// TIA Portal V20 export
// export: Created 2025-12-01T14:57:00.8344037Z, ExportSetting None, DisplayName Totally Integrated Automation Portal, DisplayVersion V20 Update 3, DisplayName TIA Portal Openness, DisplayVersion V20 Update 3, DisplayName TIA Portal Version Control Interface, DisplayVersion V20 Update 3, DisplayName STEP 7 Professional, DisplayVersion V20 Update 3, DisplayName STEP 7 Safety, DisplayVersion V20 Update 2, DisplayName WinCC Basic/Comfort/Advanced, DisplayVersion V20 Update 3, DisplayName WinCC Professional, DisplayVersion V20 Update 3, DisplayName WinCC Unified, DisplayVersion V20 Update 3
FUNCTION "FC455_TL_TR_E1_S2_Aus" : Void   // FC455, LAD
{ S7_Optimized_Access := 'FALSE' }
AUTHOR : TLigero
NAME : 20160208
VERSION : 3.5
// stored: AutoNumber false, SetENOAutomatically false
   VAR_INPUT
      Mesa : UInt;
      En_Tension : Bool;
      pHsMx_E1 : Bool;
      pHsMx_S2 : Bool;
      Termico_E1_Tx : Bool;
      Termico_S2_Tx : Bool;
      Avance_E1_Tx_Ok : Bool;
      Avance_S2_Tx_Ok : Bool;
      PosTR_E1 : Bool;
      PosTR_S2 : Bool;
      AVTF_MAnt_Mx : Bool;
      PTF_Mx_MSig : Bool;
      NXT_Avance : Bool;
      V_CNT_ApHsMx_E1 : UDInt;
      V_CNT_ApHsMx_S2 : UDInt;
      V_Paro : UDInt;
      V_TOut_Tx_Mx : UDInt;
      V_TOut_TR : UDInt;
   END_VAR
   VAR_OUTPUT
      PTF_MAnt_Mx : Bool;
      AVTF_Mx_MSig : Bool;
      NXT_Descarga_Act : Bool;
   END_VAR
   VAR_IN_OUT
      MAux_FN_Phs_E1 : Bool;
      Maux_FN_Phs_S2 : Bool;
      Mem_FN_phs_E1 : Bool;
      Mem_FN_phs_S2 : Bool;
   END_VAR
   VAR_TEMP
      Mem_CNT_Aus_Ent : Bool;
      OK_VACIADO : Bool;
      Mem_CNT_Aus_Sal : Bool;
      Aux_Parar : Bool;
      tout_atasco : Bool;
      tout_transfer : Bool;
      Mem_CNT_Tmp_Paro_Tx : Bool;
      TEMP_MA_TR_Pos_E1 : Bool;
      TEMP_MA_TR_Pos_S2 : Bool;
      ok_tension : Bool;
   END_VAR
   VAR_TEMP   // added for the SCL form of the ladder/FBD networks
      _w1 : Bool;
      _w2 : Bool;
   END_VAR
BEGIN

REGION Network 1: Marca General Error
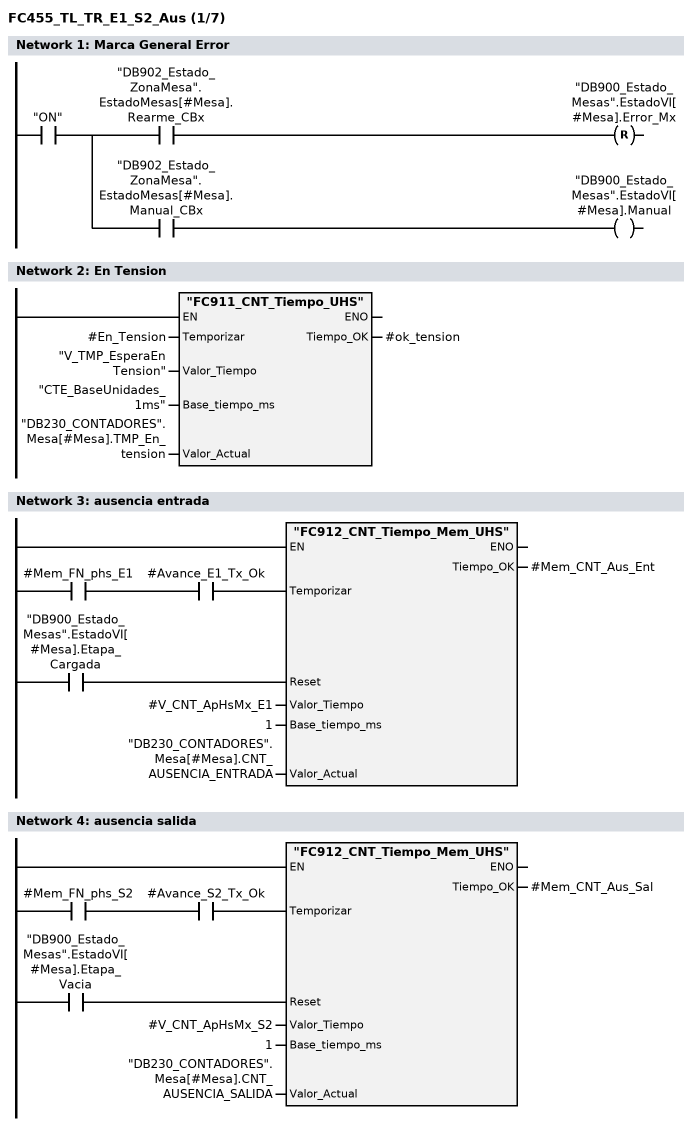
   RUNG wire#powerrail
      Contact( "ON" )
      wire#w1
      Contact( "DB902_Estado_ZonaMesa".EstadoMesas[#Mesa].Rearme_CBx )
      R_Coil( "DB900_Estado_Mesas".EstadoVI[#Mesa].Error_Mx )
   END_RUNG
   RUNG wire#w1
      Contact( "DB902_Estado_ZonaMesa".EstadoMesas[#Mesa].Manual_CBx )
      Coil( "DB900_Estado_Mesas".EstadoVI[#Mesa].Manual )
   END_RUNG
   // the same network as SCL:
   IF "ON" AND "DB902_Estado_ZonaMesa".EstadoMesas[#Mesa].Rearme_CBx THEN
       "DB900_Estado_Mesas".EstadoVI[#Mesa].Error_Mx := FALSE;
   END_IF;
   "DB900_Estado_Mesas".EstadoVI[#Mesa].Manual := "ON" AND "DB902_Estado_ZonaMesa".EstadoMesas[#Mesa].Manual_CBx;
END_REGION

REGION Network 2: En Tension
   RUNG wire#powerrail
      "FC911_CNT_Tiempo_UHS"(Temporizar := #En_Tension, Valor_Tiempo := "V_TMP_EsperaEnTension", Base_tiempo_ms := "CTE_BaseUnidades_1ms", Valor_Actual := "DB230_CONTADORES".Mesa[#Mesa].TMP_En_tension, Tiempo_OK => #ok_tension)
   END_RUNG
   // the same network as SCL:
   "FC911_CNT_Tiempo_UHS"(Temporizar := #En_Tension,
                          Valor_Tiempo := "V_TMP_EsperaEnTension",
                          Base_tiempo_ms := "CTE_BaseUnidades_1ms",
                          Valor_Actual := "DB230_CONTADORES".Mesa[#Mesa].TMP_En_tension,
                          Tiempo_OK => #ok_tension);
END_REGION

REGION Network 3: ausencia entrada
   RUNG wire#powerrail
      "FC912_CNT_Tiempo_Mem_UHS"(Temporizar := wire#w1, Reset := wire#w2, Valor_Tiempo := #V_CNT_ApHsMx_E1, Base_tiempo_ms := 1, Valor_Actual := "DB230_CONTADORES".Mesa[#Mesa].CNT_AUSENCIA_ENTRADA, Tiempo_OK => #Mem_CNT_Aus_Ent)
   END_RUNG
   RUNG wire#powerrail
      Contact( #Mem_FN_phs_E1 )
      Contact( #Avance_E1_Tx_Ok )
   END_RUNG wire#w1
   RUNG wire#powerrail
      Contact( "DB900_Estado_Mesas".EstadoVI[#Mesa].Etapa_Cargada )
   END_RUNG wire#w2
   // the same network as SCL:
   "FC912_CNT_Tiempo_Mem_UHS"(Temporizar := #Mem_FN_phs_E1 AND #Avance_E1_Tx_Ok,
                           Reset := "DB900_Estado_Mesas".EstadoVI[#Mesa].Etapa_Cargada,
                           Valor_Tiempo := #V_CNT_ApHsMx_E1,
                           Base_tiempo_ms := 1,
                           Valor_Actual := "DB230_CONTADORES".Mesa[#Mesa].CNT_AUSENCIA_ENTRADA,
                           Tiempo_OK => #Mem_CNT_Aus_Ent);
END_REGION

REGION Network 4: ausencia salida
   RUNG wire#powerrail
      "FC912_CNT_Tiempo_Mem_UHS"(Temporizar := wire#w1, Reset := wire#w2, Valor_Tiempo := #V_CNT_ApHsMx_S2, Base_tiempo_ms := 1, Valor_Actual := "DB230_CONTADORES".Mesa[#Mesa].CNT_AUSENCIA_SALIDA, Tiempo_OK => #Mem_CNT_Aus_Sal)
   END_RUNG
   RUNG wire#powerrail
      Contact( #Mem_FN_phs_S2 )
      Contact( #Avance_S2_Tx_Ok )
   END_RUNG wire#w1
   RUNG wire#powerrail
      Contact( "DB900_Estado_Mesas".EstadoVI[#Mesa].Etapa_Vacia )
   END_RUNG wire#w2
   // the same network as SCL:
   "FC912_CNT_Tiempo_Mem_UHS"(Temporizar := #Mem_FN_phs_S2 AND #Avance_S2_Tx_Ok,
                           Reset := "DB900_Estado_Mesas".EstadoVI[#Mesa].Etapa_Vacia,
                           Valor_Tiempo := #V_CNT_ApHsMx_S2,
                           Base_tiempo_ms := 1,
                           Valor_Actual := "DB230_CONTADORES".Mesa[#Mesa].CNT_AUSENCIA_SALIDA,
                           Tiempo_OK => #Mem_CNT_Aus_Sal);
END_REGION

REGION Network 5: MEMORIAS DE FLANCOS
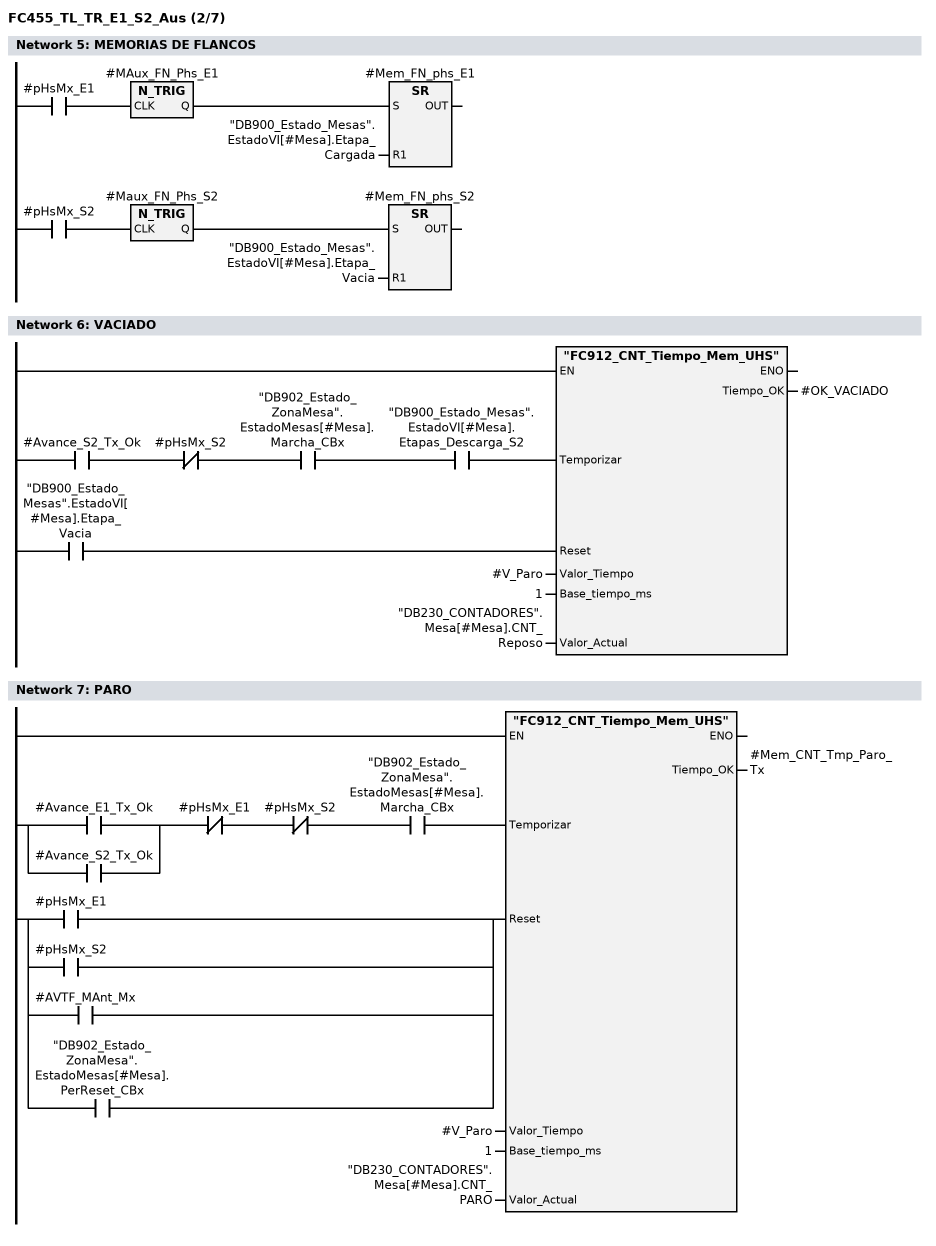
   RUNG wire#powerrail
      Contact( #pHsMx_E1 )
      N_Trig( #MAux_FN_Phs_E1 )
      S_SR(operand := #Mem_FN_phs_E1, r1 := "DB900_Estado_Mesas".EstadoVI[#Mesa].Etapa_Cargada)
   END_RUNG
   RUNG wire#powerrail
      Contact( #pHsMx_S2 )
      N_Trig( #Maux_FN_Phs_S2 )
      S_SR(operand := #Mem_FN_phs_S2, r1 := "DB900_Estado_Mesas".EstadoVI[#Mesa].Etapa_Vacia)
   END_RUNG
   // the same network as SCL:
   #_w1 := NOT #pHsMx_E1 AND #MAux_FN_Phs_E1;   // falling edge
   #MAux_FN_Phs_E1 := #pHsMx_E1;
   IF #_w1 THEN
       #Mem_FN_phs_E1 := TRUE;   // SR flip-flop
   END_IF;
   IF "DB900_Estado_Mesas".EstadoVI[#Mesa].Etapa_Cargada THEN #Mem_FN_phs_E1 := FALSE; END_IF;
   #_w2 := NOT #pHsMx_S2 AND #Maux_FN_Phs_S2;   // falling edge
   #Maux_FN_Phs_S2 := #pHsMx_S2;
   IF #_w2 THEN
       #Mem_FN_phs_S2 := TRUE;   // SR flip-flop
   END_IF;
   IF "DB900_Estado_Mesas".EstadoVI[#Mesa].Etapa_Vacia THEN #Mem_FN_phs_S2 := FALSE; END_IF;
END_REGION

REGION Network 6: VACIADO
   RUNG wire#powerrail
      "FC912_CNT_Tiempo_Mem_UHS"(Temporizar := wire#w1, Reset := wire#w2, Valor_Tiempo := #V_Paro, Base_tiempo_ms := 1, Valor_Actual := "DB230_CONTADORES".Mesa[#Mesa].CNT_Reposo, Tiempo_OK => #OK_VACIADO)
   END_RUNG
   RUNG wire#powerrail
      Contact( #Avance_S2_Tx_Ok )
      I_Contact( #pHsMx_S2 )
      Contact( "DB902_Estado_ZonaMesa".EstadoMesas[#Mesa].Marcha_CBx )
      Contact( "DB900_Estado_Mesas".EstadoVI[#Mesa].Etapas_Descarga_S2 )
   END_RUNG wire#w1
   RUNG wire#powerrail
      Contact( "DB900_Estado_Mesas".EstadoVI[#Mesa].Etapa_Vacia )
   END_RUNG wire#w2
   // the same network as SCL:
   "FC912_CNT_Tiempo_Mem_UHS"(Temporizar := #Avance_S2_Tx_Ok AND NOT #pHsMx_S2 AND "DB902_Estado_ZonaMesa".EstadoMesas[#Mesa].Marcha_CBx AND "DB900_Estado_Mesas".EstadoVI[#Mesa].Etapas_Descarga_S2,
                           Reset := "DB900_Estado_Mesas".EstadoVI[#Mesa].Etapa_Vacia,
                           Valor_Tiempo := #V_Paro,
                           Base_tiempo_ms := 1,
                           Valor_Actual := "DB230_CONTADORES".Mesa[#Mesa].CNT_Reposo,
                           Tiempo_OK => #OK_VACIADO);
END_REGION

REGION Network 7: PARO
   RUNG wire#powerrail
      "FC912_CNT_Tiempo_Mem_UHS"(Temporizar := wire#w2, Reset := wire#w3, Valor_Tiempo := #V_Paro, Base_tiempo_ms := 1, Valor_Actual := "DB230_CONTADORES".Mesa[#Mesa].CNT_PARO, Tiempo_OK => #Mem_CNT_Tmp_Paro_Tx)
   END_RUNG
   RUNG wire#powerrail
      Contact( #Avance_E1_Tx_Ok )
      wire#w1
      I_Contact( #pHsMx_E1 )
      I_Contact( #pHsMx_S2 )
      Contact( "DB902_Estado_ZonaMesa".EstadoMesas[#Mesa].Marcha_CBx )
   END_RUNG wire#w2
   RUNG wire#powerrail
      Contact( #Avance_S2_Tx_Ok )
   END_RUNG wire#w1
   RUNG wire#powerrail
      Contact( #pHsMx_E1 )
   END_RUNG wire#w3
   RUNG wire#powerrail
      Contact( #pHsMx_S2 )
   END_RUNG wire#w3
   RUNG wire#powerrail
      Contact( #AVTF_MAnt_Mx )
   END_RUNG wire#w3
   RUNG wire#powerrail
      Contact( "DB902_Estado_ZonaMesa".EstadoMesas[#Mesa].PerReset_CBx )
   END_RUNG wire#w3
   // the same network as SCL:
   "FC912_CNT_Tiempo_Mem_UHS"(Temporizar := (#Avance_E1_Tx_Ok OR #Avance_S2_Tx_Ok) AND NOT #pHsMx_E1 AND NOT #pHsMx_S2 AND "DB902_Estado_ZonaMesa".EstadoMesas[#Mesa].Marcha_CBx,
                           Reset := #pHsMx_E1 OR #pHsMx_S2 OR #AVTF_MAnt_Mx OR "DB902_Estado_ZonaMesa".EstadoMesas[#Mesa].PerReset_CBx,
                           Valor_Tiempo := #V_Paro,
                           Base_tiempo_ms := 1,
                           Valor_Actual := "DB230_CONTADORES".Mesa[#Mesa].CNT_PARO,
                           Tiempo_OK => #Mem_CNT_Tmp_Paro_Tx);
END_REGION

REGION Network 8: Etapa MESA CARGADA
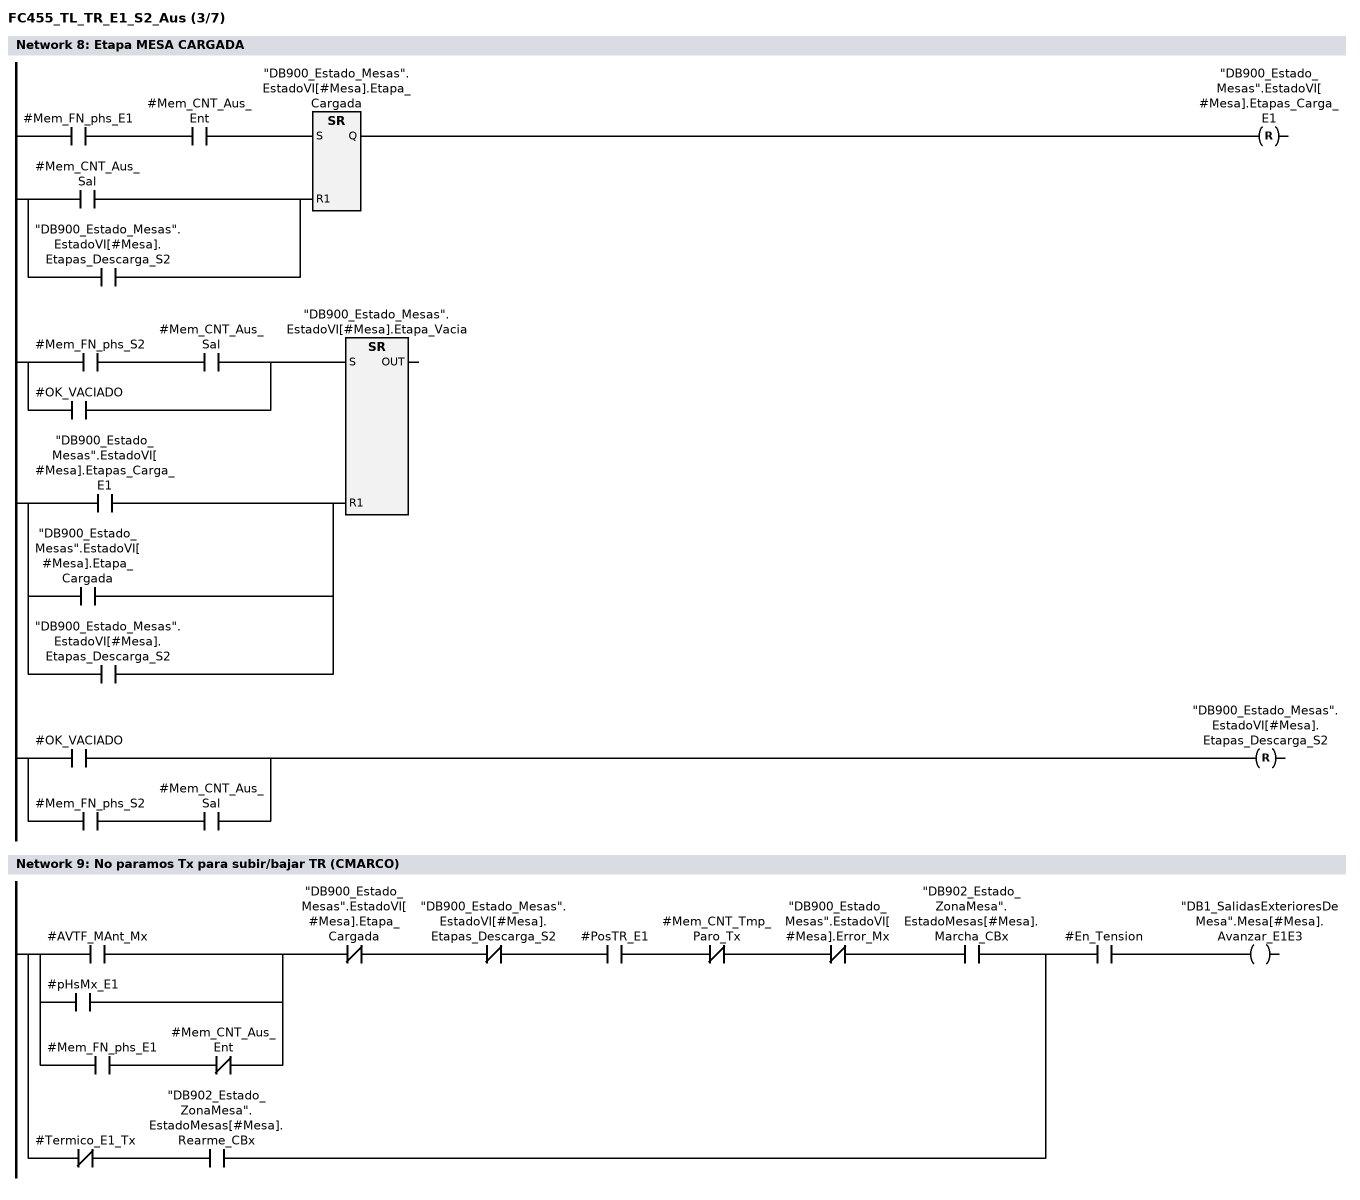
   RUNG wire#powerrail
      Contact( #Mem_FN_phs_E1 )
      Contact( #Mem_CNT_Aus_Ent )
      S_SR(operand := "DB900_Estado_Mesas".EstadoVI[#Mesa].Etapa_Cargada, r1 := wire#w1)
      R_Coil( "DB900_Estado_Mesas".EstadoVI[#Mesa].Etapas_Carga_E1 )
   END_RUNG
   RUNG wire#powerrail
      Contact( #Mem_CNT_Aus_Sal )
   END_RUNG wire#w1
   RUNG wire#powerrail
      Contact( "DB900_Estado_Mesas".EstadoVI[#Mesa].Etapas_Descarga_S2 )
   END_RUNG wire#w1
   RUNG wire#powerrail
      Contact( #Mem_FN_phs_S2 )
      Contact( #Mem_CNT_Aus_Sal )
      wire#w2
      S_SR(operand := "DB900_Estado_Mesas".EstadoVI[#Mesa].Etapa_Vacia, r1 := wire#w3)
   END_RUNG
   RUNG wire#powerrail
      Contact( #OK_VACIADO )
   END_RUNG wire#w2
   RUNG wire#powerrail
      Contact( "DB900_Estado_Mesas".EstadoVI[#Mesa].Etapas_Carga_E1 )
   END_RUNG wire#w3
   RUNG wire#powerrail
      Contact( "DB900_Estado_Mesas".EstadoVI[#Mesa].Etapa_Cargada )
   END_RUNG wire#w3
   RUNG wire#powerrail
      Contact( "DB900_Estado_Mesas".EstadoVI[#Mesa].Etapas_Descarga_S2 )
   END_RUNG wire#w3
   RUNG wire#powerrail
      Contact( #OK_VACIADO )
      wire#w4
      R_Coil( "DB900_Estado_Mesas".EstadoVI[#Mesa].Etapas_Descarga_S2 )
   END_RUNG
   RUNG wire#powerrail
      Contact( #Mem_FN_phs_S2 )
      Contact( #Mem_CNT_Aus_Sal )
   END_RUNG wire#w4
   // the same network as SCL:
   #_w1 := #Mem_CNT_Aus_Sal OR "DB900_Estado_Mesas".EstadoVI[#Mesa].Etapas_Descarga_S2;
   IF #Mem_FN_phs_E1 AND #Mem_CNT_Aus_Ent THEN
       "DB900_Estado_Mesas".EstadoVI[#Mesa].Etapa_Cargada := TRUE;   // SR flip-flop
   END_IF;
   IF #_w1 THEN "DB900_Estado_Mesas".EstadoVI[#Mesa].Etapa_Cargada := FALSE; END_IF;
   IF "DB900_Estado_Mesas".EstadoVI[#Mesa].Etapa_Cargada THEN
       "DB900_Estado_Mesas".EstadoVI[#Mesa].Etapas_Carga_E1 := FALSE;
   END_IF;
   #_w2 := "DB900_Estado_Mesas".EstadoVI[#Mesa].Etapas_Carga_E1 OR "DB900_Estado_Mesas".EstadoVI[#Mesa].Etapa_Cargada OR "DB900_Estado_Mesas".EstadoVI[#Mesa].Etapas_Descarga_S2;
   IF (#Mem_FN_phs_S2 AND #Mem_CNT_Aus_Sal) OR #OK_VACIADO THEN
       "DB900_Estado_Mesas".EstadoVI[#Mesa].Etapa_Vacia := TRUE;   // SR flip-flop
   END_IF;
   IF #_w2 THEN "DB900_Estado_Mesas".EstadoVI[#Mesa].Etapa_Vacia := FALSE; END_IF;
   IF #OK_VACIADO OR (#Mem_FN_phs_S2 AND #Mem_CNT_Aus_Sal) THEN
       "DB900_Estado_Mesas".EstadoVI[#Mesa].Etapas_Descarga_S2 := FALSE;
   END_IF;
END_REGION

REGION Network 9: No paramos Tx para subir/bajar TR (CMARCO)
   RUNG wire#powerrail
      Contact( #AVTF_MAnt_Mx )
      wire#w1
      I_Contact( "DB900_Estado_Mesas".EstadoVI[#Mesa].Etapa_Cargada )
      I_Contact( "DB900_Estado_Mesas".EstadoVI[#Mesa].Etapas_Descarga_S2 )
      Contact( #PosTR_E1 )
      I_Contact( #Mem_CNT_Tmp_Paro_Tx )
      I_Contact( "DB900_Estado_Mesas".EstadoVI[#Mesa].Error_Mx )
      Contact( "DB902_Estado_ZonaMesa".EstadoMesas[#Mesa].Marcha_CBx )
      wire#w2
      Contact( #En_Tension )
      Coil( "DB1_SalidasExterioresDeMesa".Mesa[#Mesa].Avanzar_E1E3 )
   END_RUNG
   RUNG wire#powerrail
      Contact( #pHsMx_E1 )
   END_RUNG wire#w1
   RUNG wire#powerrail
      Contact( #Mem_FN_phs_E1 )
      I_Contact( #Mem_CNT_Aus_Ent )
   END_RUNG wire#w1
   RUNG wire#powerrail
      I_Contact( #Termico_E1_Tx )
      Contact( "DB902_Estado_ZonaMesa".EstadoMesas[#Mesa].Rearme_CBx )
   END_RUNG wire#w2
   // the same network as SCL:
   "DB1_SalidasExterioresDeMesa".Mesa[#Mesa].Avanzar_E1E3 := (((#AVTF_MAnt_Mx OR #pHsMx_E1 OR (#Mem_FN_phs_E1 AND NOT #Mem_CNT_Aus_Ent)) AND NOT "DB900_Estado_Mesas".EstadoVI[#Mesa].Etapa_Cargada AND NOT "DB900_Estado_Mesas".EstadoVI[#Mesa].Etapas_Descarga_S2 AND #PosTR_E1 AND NOT #Mem_CNT_Tmp_Paro_Tx AND NOT "DB900_Estado_Mesas".EstadoVI[#Mesa].Error_Mx AND "DB902_Estado_ZonaMesa".EstadoMesas[#Mesa].Marcha_CBx) OR (NOT #Termico_E1_Tx AND "DB902_Estado_ZonaMesa".EstadoMesas[#Mesa].Rearme_CBx)) AND #En_Tension;
END_REGION

REGION Network 10: Quito el forzar paroTx (MA 02/06/08)
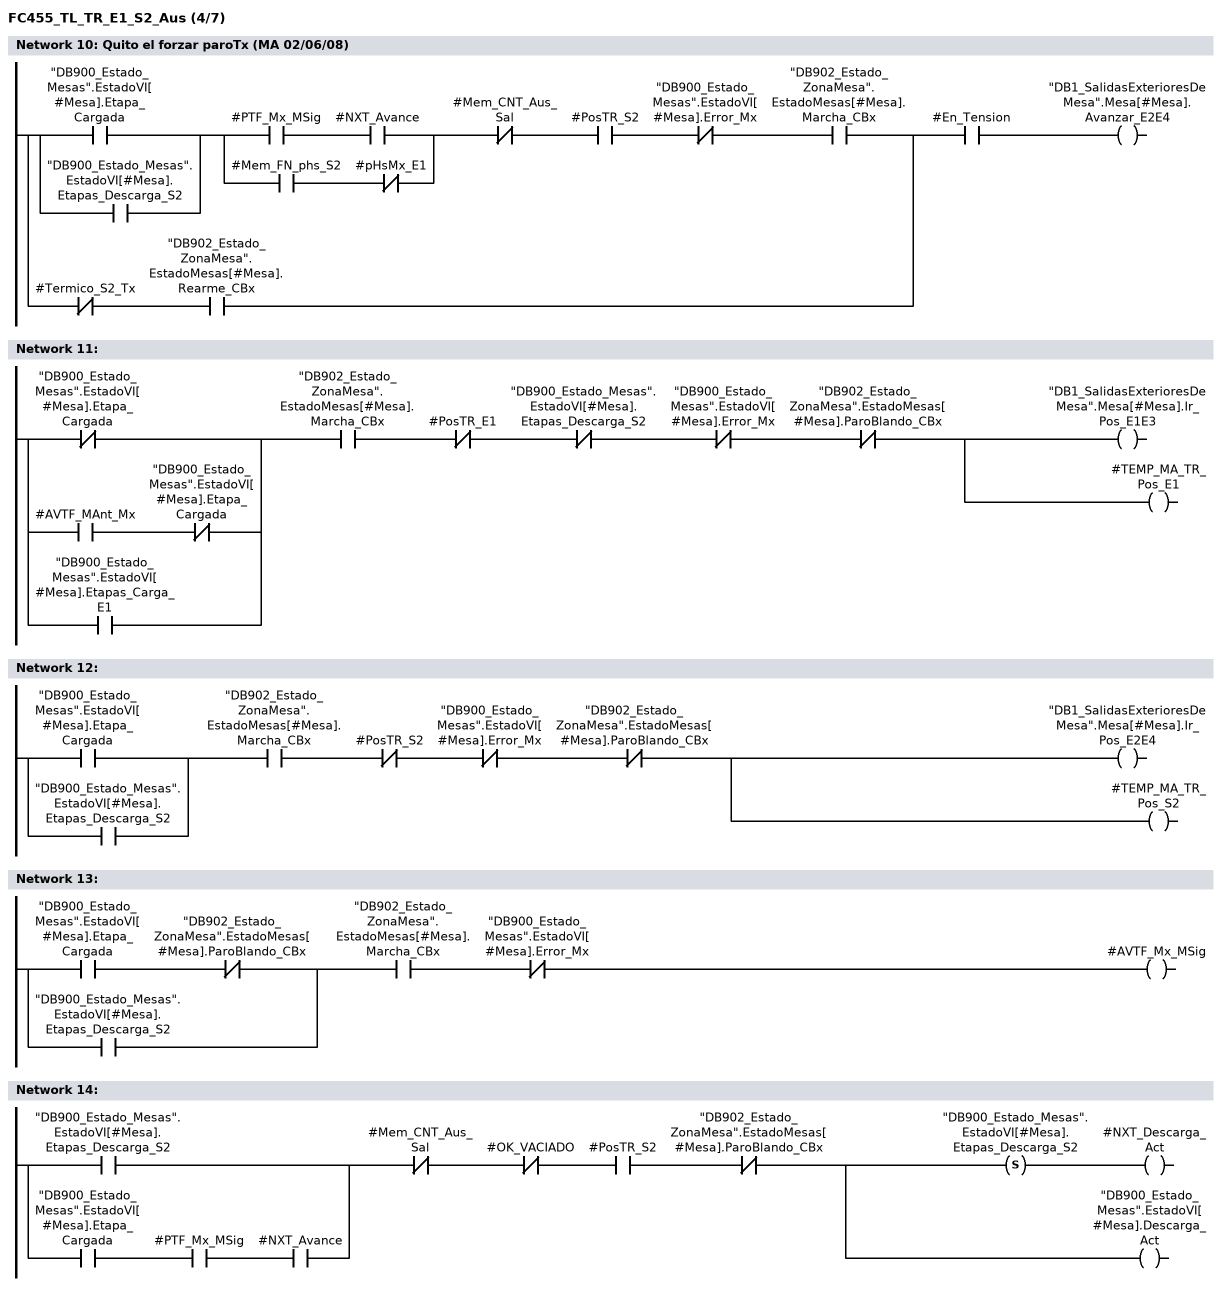
   RUNG wire#powerrail
      Contact( "DB900_Estado_Mesas".EstadoVI[#Mesa].Etapa_Cargada )
      wire#w1
      Contact( #PTF_Mx_MSig )
      Contact( #NXT_Avance )
      wire#w2
      I_Contact( #Mem_CNT_Aus_Sal )
      Contact( #PosTR_S2 )
      I_Contact( "DB900_Estado_Mesas".EstadoVI[#Mesa].Error_Mx )
      Contact( "DB902_Estado_ZonaMesa".EstadoMesas[#Mesa].Marcha_CBx )
      wire#w3
      Contact( #En_Tension )
      Coil( "DB1_SalidasExterioresDeMesa".Mesa[#Mesa].Avanzar_E2E4 )
   END_RUNG
   RUNG wire#powerrail
      Contact( "DB900_Estado_Mesas".EstadoVI[#Mesa].Etapas_Descarga_S2 )
   END_RUNG wire#w1
   RUNG wire#w1
      Contact( #Mem_FN_phs_S2 )
      I_Contact( #pHsMx_E1 )
   END_RUNG wire#w2
   RUNG wire#powerrail
      I_Contact( #Termico_S2_Tx )
      Contact( "DB902_Estado_ZonaMesa".EstadoMesas[#Mesa].Rearme_CBx )
   END_RUNG wire#w3
   // the same network as SCL:
   "DB1_SalidasExterioresDeMesa".Mesa[#Mesa].Avanzar_E2E4 := ((("DB900_Estado_Mesas".EstadoVI[#Mesa].Etapa_Cargada OR "DB900_Estado_Mesas".EstadoVI[#Mesa].Etapas_Descarga_S2) AND ((#PTF_Mx_MSig AND #NXT_Avance) OR (#Mem_FN_phs_S2 AND NOT #pHsMx_E1)) AND NOT #Mem_CNT_Aus_Sal AND #PosTR_S2 AND NOT "DB900_Estado_Mesas".EstadoVI[#Mesa].Error_Mx AND "DB902_Estado_ZonaMesa".EstadoMesas[#Mesa].Marcha_CBx) OR (NOT #Termico_S2_Tx AND "DB902_Estado_ZonaMesa".EstadoMesas[#Mesa].Rearme_CBx)) AND #En_Tension;
END_REGION

REGION Network 11
   RUNG wire#powerrail
      I_Contact( "DB900_Estado_Mesas".EstadoVI[#Mesa].Etapa_Cargada )
      wire#w1
      Contact( "DB902_Estado_ZonaMesa".EstadoMesas[#Mesa].Marcha_CBx )
      I_Contact( #PosTR_E1 )
      I_Contact( "DB900_Estado_Mesas".EstadoVI[#Mesa].Etapas_Descarga_S2 )
      I_Contact( "DB900_Estado_Mesas".EstadoVI[#Mesa].Error_Mx )
      I_Contact( "DB902_Estado_ZonaMesa".EstadoMesas[#Mesa].ParoBlando_CBx )
      wire#w2
      Coil( "DB1_SalidasExterioresDeMesa".Mesa[#Mesa].Ir_Pos_E1E3 )
   END_RUNG
   RUNG wire#powerrail
      Contact( #AVTF_MAnt_Mx )
      I_Contact( "DB900_Estado_Mesas".EstadoVI[#Mesa].Etapa_Cargada )
   END_RUNG wire#w1
   RUNG wire#powerrail
      Contact( "DB900_Estado_Mesas".EstadoVI[#Mesa].Etapas_Carga_E1 )
   END_RUNG wire#w1
   RUNG wire#w2
      Coil( #TEMP_MA_TR_Pos_E1 )
   END_RUNG
   // the same network as SCL:
   #_w1 := (NOT "DB900_Estado_Mesas".EstadoVI[#Mesa].Etapa_Cargada OR (#AVTF_MAnt_Mx AND NOT "DB900_Estado_Mesas".EstadoVI[#Mesa].Etapa_Cargada) OR "DB900_Estado_Mesas".EstadoVI[#Mesa].Etapas_Carga_E1) AND "DB902_Estado_ZonaMesa".EstadoMesas[#Mesa].Marcha_CBx AND NOT #PosTR_E1 AND NOT "DB900_Estado_Mesas".EstadoVI[#Mesa].Etapas_Descarga_S2 AND NOT "DB900_Estado_Mesas".EstadoVI[#Mesa].Error_Mx AND NOT "DB902_Estado_ZonaMesa".EstadoMesas[#Mesa].ParoBlando_CBx;
   "DB1_SalidasExterioresDeMesa".Mesa[#Mesa].Ir_Pos_E1E3 := (NOT "DB900_Estado_Mesas".EstadoVI[#Mesa].Etapa_Cargada OR (#AVTF_MAnt_Mx AND NOT "DB900_Estado_Mesas".EstadoVI[#Mesa].Etapa_Cargada) OR "DB900_Estado_Mesas".EstadoVI[#Mesa].Etapas_Carga_E1) AND "DB902_Estado_ZonaMesa".EstadoMesas[#Mesa].Marcha_CBx AND NOT #PosTR_E1 AND NOT "DB900_Estado_Mesas".EstadoVI[#Mesa].Etapas_Descarga_S2 AND NOT "DB900_Estado_Mesas".EstadoVI[#Mesa].Error_Mx AND NOT "DB902_Estado_ZonaMesa".EstadoMesas[#Mesa].ParoBlando_CBx;
   #TEMP_MA_TR_Pos_E1 := #_w1;
END_REGION

REGION Network 12
   RUNG wire#powerrail
      Contact( "DB900_Estado_Mesas".EstadoVI[#Mesa].Etapa_Cargada )
      wire#w1
      Contact( "DB902_Estado_ZonaMesa".EstadoMesas[#Mesa].Marcha_CBx )
      I_Contact( #PosTR_S2 )
      I_Contact( "DB900_Estado_Mesas".EstadoVI[#Mesa].Error_Mx )
      I_Contact( "DB902_Estado_ZonaMesa".EstadoMesas[#Mesa].ParoBlando_CBx )
      wire#w2
      Coil( "DB1_SalidasExterioresDeMesa".Mesa[#Mesa].Ir_Pos_E2E4 )
   END_RUNG
   RUNG wire#powerrail
      Contact( "DB900_Estado_Mesas".EstadoVI[#Mesa].Etapas_Descarga_S2 )
   END_RUNG wire#w1
   RUNG wire#w2
      Coil( #TEMP_MA_TR_Pos_S2 )
   END_RUNG
   // the same network as SCL:
   #_w1 := ("DB900_Estado_Mesas".EstadoVI[#Mesa].Etapa_Cargada OR "DB900_Estado_Mesas".EstadoVI[#Mesa].Etapas_Descarga_S2) AND "DB902_Estado_ZonaMesa".EstadoMesas[#Mesa].Marcha_CBx AND NOT #PosTR_S2 AND NOT "DB900_Estado_Mesas".EstadoVI[#Mesa].Error_Mx AND NOT "DB902_Estado_ZonaMesa".EstadoMesas[#Mesa].ParoBlando_CBx;
   "DB1_SalidasExterioresDeMesa".Mesa[#Mesa].Ir_Pos_E2E4 := ("DB900_Estado_Mesas".EstadoVI[#Mesa].Etapa_Cargada OR "DB900_Estado_Mesas".EstadoVI[#Mesa].Etapas_Descarga_S2) AND "DB902_Estado_ZonaMesa".EstadoMesas[#Mesa].Marcha_CBx AND NOT #PosTR_S2 AND NOT "DB900_Estado_Mesas".EstadoVI[#Mesa].Error_Mx AND NOT "DB902_Estado_ZonaMesa".EstadoMesas[#Mesa].ParoBlando_CBx;
   #TEMP_MA_TR_Pos_S2 := #_w1;
END_REGION

REGION Network 13
   RUNG wire#powerrail
      Contact( "DB900_Estado_Mesas".EstadoVI[#Mesa].Etapa_Cargada )
      I_Contact( "DB902_Estado_ZonaMesa".EstadoMesas[#Mesa].ParoBlando_CBx )
      wire#w1
      Contact( "DB902_Estado_ZonaMesa".EstadoMesas[#Mesa].Marcha_CBx )
      I_Contact( "DB900_Estado_Mesas".EstadoVI[#Mesa].Error_Mx )
      Coil( #AVTF_Mx_MSig )
   END_RUNG
   RUNG wire#powerrail
      Contact( "DB900_Estado_Mesas".EstadoVI[#Mesa].Etapas_Descarga_S2 )
   END_RUNG wire#w1
   // the same network as SCL:
   #AVTF_Mx_MSig := (("DB900_Estado_Mesas".EstadoVI[#Mesa].Etapa_Cargada AND NOT "DB902_Estado_ZonaMesa".EstadoMesas[#Mesa].ParoBlando_CBx) OR "DB900_Estado_Mesas".EstadoVI[#Mesa].Etapas_Descarga_S2) AND "DB902_Estado_ZonaMesa".EstadoMesas[#Mesa].Marcha_CBx AND NOT "DB900_Estado_Mesas".EstadoVI[#Mesa].Error_Mx;
END_REGION

REGION Network 14
   RUNG wire#powerrail
      Contact( "DB900_Estado_Mesas".EstadoVI[#Mesa].Etapas_Descarga_S2 )
      wire#w1
      I_Contact( #Mem_CNT_Aus_Sal )
      I_Contact( #OK_VACIADO )
      Contact( #PosTR_S2 )
      I_Contact( "DB902_Estado_ZonaMesa".EstadoMesas[#Mesa].ParoBlando_CBx )
      wire#w2
      S_Coil( "DB900_Estado_Mesas".EstadoVI[#Mesa].Etapas_Descarga_S2 )
      Coil( #NXT_Descarga_Act )
   END_RUNG
   RUNG wire#powerrail
      Contact( "DB900_Estado_Mesas".EstadoVI[#Mesa].Etapa_Cargada )
      Contact( #PTF_Mx_MSig )
      Contact( #NXT_Avance )
   END_RUNG wire#w1
   RUNG wire#w2
      Coil( "DB900_Estado_Mesas".EstadoVI[#Mesa].Descarga_Act )
   END_RUNG
   // the same network as SCL:
   #_w1 := ("DB900_Estado_Mesas".EstadoVI[#Mesa].Etapas_Descarga_S2 OR ("DB900_Estado_Mesas".EstadoVI[#Mesa].Etapa_Cargada AND #PTF_Mx_MSig AND #NXT_Avance)) AND NOT #Mem_CNT_Aus_Sal AND NOT #OK_VACIADO AND #PosTR_S2 AND NOT "DB902_Estado_ZonaMesa".EstadoMesas[#Mesa].ParoBlando_CBx;
   IF #_w1 THEN "DB900_Estado_Mesas".EstadoVI[#Mesa].Etapas_Descarga_S2 := TRUE; END_IF;
   #NXT_Descarga_Act := #_w1;
   "DB900_Estado_Mesas".EstadoVI[#Mesa].Descarga_Act := #_w1;
END_REGION

REGION Network 15
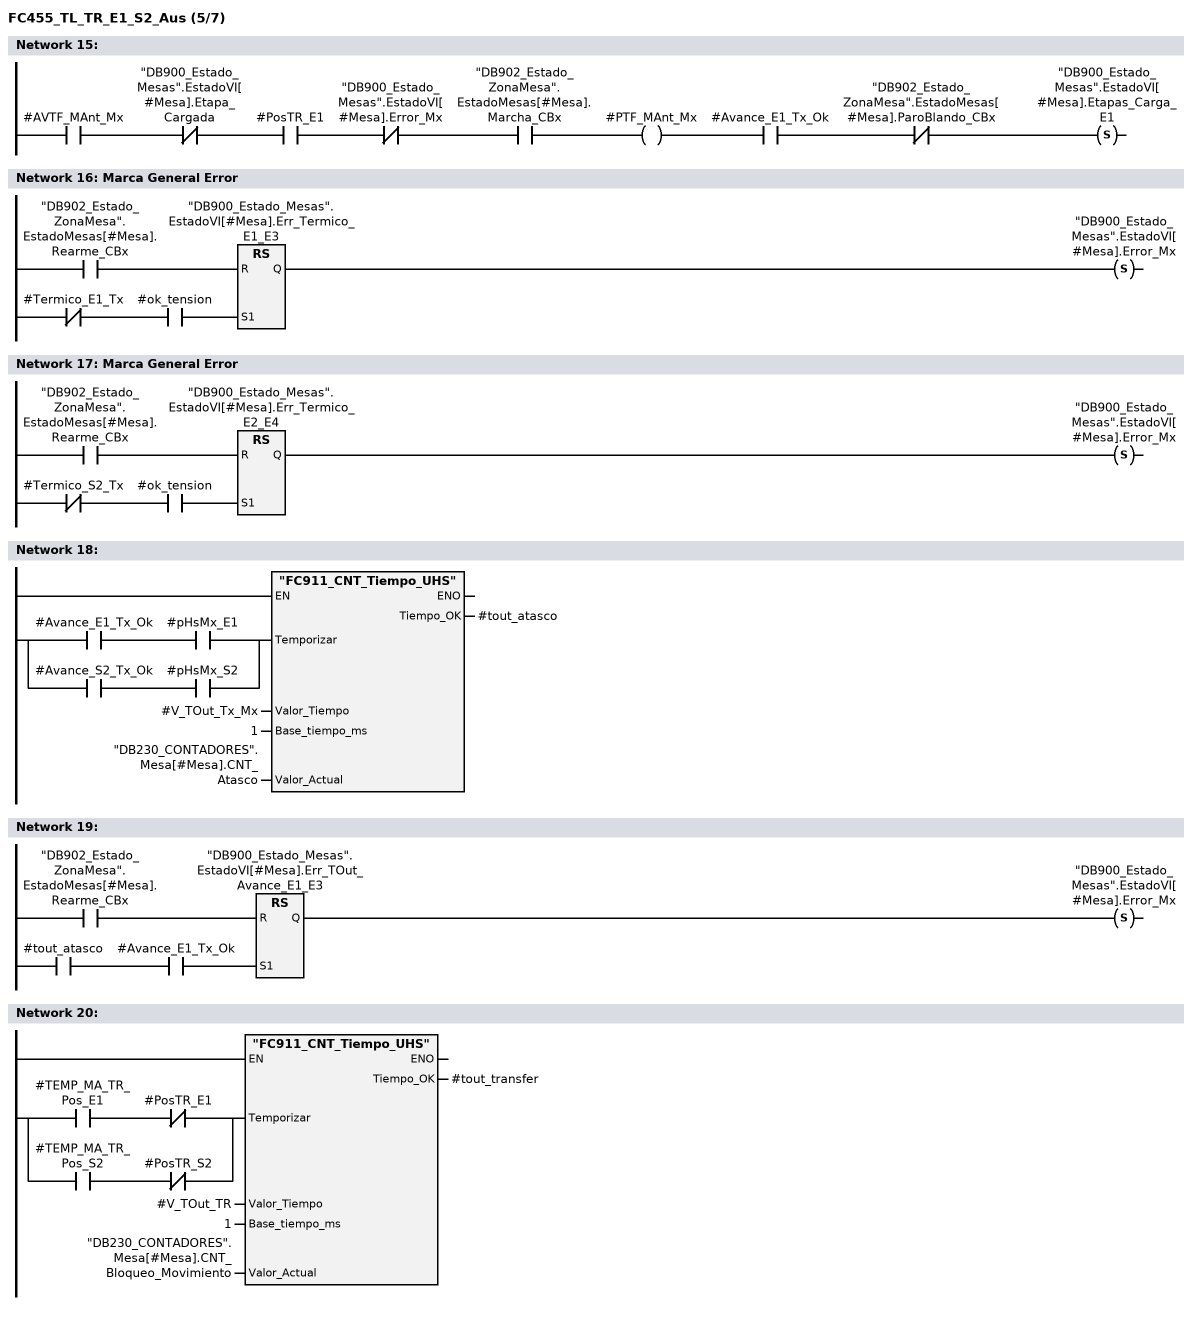
   RUNG wire#powerrail
      Contact( #AVTF_MAnt_Mx )
      I_Contact( "DB900_Estado_Mesas".EstadoVI[#Mesa].Etapa_Cargada )
      Contact( #PosTR_E1 )
      I_Contact( "DB900_Estado_Mesas".EstadoVI[#Mesa].Error_Mx )
      Contact( "DB902_Estado_ZonaMesa".EstadoMesas[#Mesa].Marcha_CBx )
      Coil( #PTF_MAnt_Mx )
      Contact( #Avance_E1_Tx_Ok )
      I_Contact( "DB902_Estado_ZonaMesa".EstadoMesas[#Mesa].ParoBlando_CBx )
      S_Coil( "DB900_Estado_Mesas".EstadoVI[#Mesa].Etapas_Carga_E1 )
   END_RUNG
   // the same network as SCL:
   #PTF_MAnt_Mx := #AVTF_MAnt_Mx AND NOT "DB900_Estado_Mesas".EstadoVI[#Mesa].Etapa_Cargada AND #PosTR_E1 AND NOT "DB900_Estado_Mesas".EstadoVI[#Mesa].Error_Mx AND "DB902_Estado_ZonaMesa".EstadoMesas[#Mesa].Marcha_CBx;
   IF #PTF_MAnt_Mx AND #Avance_E1_Tx_Ok AND NOT "DB902_Estado_ZonaMesa".EstadoMesas[#Mesa].ParoBlando_CBx THEN
       "DB900_Estado_Mesas".EstadoVI[#Mesa].Etapas_Carga_E1 := TRUE;
   END_IF;
END_REGION

REGION Network 16: Marca General Error
   RUNG wire#powerrail
      Contact( "DB902_Estado_ZonaMesa".EstadoMesas[#Mesa].Rearme_CBx )
      S_RS(operand := "DB900_Estado_Mesas".EstadoVI[#Mesa].Err_Termico_E1_E3, s1 := wire#w1)
      S_Coil( "DB900_Estado_Mesas".EstadoVI[#Mesa].Error_Mx )
   END_RUNG
   RUNG wire#powerrail
      I_Contact( #Termico_E1_Tx )
      Contact( #ok_tension )
   END_RUNG wire#w1
   // the same network as SCL:
   IF "DB902_Estado_ZonaMesa".EstadoMesas[#Mesa].Rearme_CBx THEN
       "DB900_Estado_Mesas".EstadoVI[#Mesa].Err_Termico_E1_E3 := FALSE;   // RS flip-flop
   END_IF;
   IF NOT #Termico_E1_Tx AND #ok_tension THEN
       "DB900_Estado_Mesas".EstadoVI[#Mesa].Err_Termico_E1_E3 := TRUE;
   END_IF;
   IF "DB900_Estado_Mesas".EstadoVI[#Mesa].Err_Termico_E1_E3 THEN
       "DB900_Estado_Mesas".EstadoVI[#Mesa].Error_Mx := TRUE;
   END_IF;
END_REGION

REGION Network 17: Marca General Error
   RUNG wire#powerrail
      Contact( "DB902_Estado_ZonaMesa".EstadoMesas[#Mesa].Rearme_CBx )
      S_RS(operand := "DB900_Estado_Mesas".EstadoVI[#Mesa].Err_Termico_E2_E4, s1 := wire#w1)
      S_Coil( "DB900_Estado_Mesas".EstadoVI[#Mesa].Error_Mx )
   END_RUNG
   RUNG wire#powerrail
      I_Contact( #Termico_S2_Tx )
      Contact( #ok_tension )
   END_RUNG wire#w1
   // the same network as SCL:
   IF "DB902_Estado_ZonaMesa".EstadoMesas[#Mesa].Rearme_CBx THEN
       "DB900_Estado_Mesas".EstadoVI[#Mesa].Err_Termico_E2_E4 := FALSE;   // RS flip-flop
   END_IF;
   IF NOT #Termico_S2_Tx AND #ok_tension THEN
       "DB900_Estado_Mesas".EstadoVI[#Mesa].Err_Termico_E2_E4 := TRUE;
   END_IF;
   IF "DB900_Estado_Mesas".EstadoVI[#Mesa].Err_Termico_E2_E4 THEN
       "DB900_Estado_Mesas".EstadoVI[#Mesa].Error_Mx := TRUE;
   END_IF;
END_REGION

REGION Network 18
   RUNG wire#powerrail
      "FC911_CNT_Tiempo_UHS"(Temporizar := wire#w1, Valor_Tiempo := #V_TOut_Tx_Mx, Base_tiempo_ms := 1, Valor_Actual := "DB230_CONTADORES".Mesa[#Mesa].CNT_Atasco, Tiempo_OK => #tout_atasco)
   END_RUNG
   RUNG wire#powerrail
      Contact( #Avance_E1_Tx_Ok )
      Contact( #pHsMx_E1 )
   END_RUNG wire#w1
   RUNG wire#powerrail
      Contact( #Avance_S2_Tx_Ok )
      Contact( #pHsMx_S2 )
   END_RUNG wire#w1
   // the same network as SCL:
   "FC911_CNT_Tiempo_UHS"(Temporizar := (#Avance_E1_Tx_Ok AND #pHsMx_E1) OR (#Avance_S2_Tx_Ok AND #pHsMx_S2),
                          Valor_Tiempo := #V_TOut_Tx_Mx,
                          Base_tiempo_ms := 1,
                          Valor_Actual := "DB230_CONTADORES".Mesa[#Mesa].CNT_Atasco,
                          Tiempo_OK => #tout_atasco);
END_REGION

REGION Network 19
   RUNG wire#powerrail
      Contact( "DB902_Estado_ZonaMesa".EstadoMesas[#Mesa].Rearme_CBx )
      S_RS(operand := "DB900_Estado_Mesas".EstadoVI[#Mesa].Err_TOut_Avance_E1_E3, s1 := wire#w1)
      S_Coil( "DB900_Estado_Mesas".EstadoVI[#Mesa].Error_Mx )
   END_RUNG
   RUNG wire#powerrail
      Contact( #tout_atasco )
      Contact( #Avance_E1_Tx_Ok )
   END_RUNG wire#w1
   // the same network as SCL:
   IF "DB902_Estado_ZonaMesa".EstadoMesas[#Mesa].Rearme_CBx THEN
       "DB900_Estado_Mesas".EstadoVI[#Mesa].Err_TOut_Avance_E1_E3 := FALSE;   // RS flip-flop
   END_IF;
   IF #tout_atasco AND #Avance_E1_Tx_Ok THEN
       "DB900_Estado_Mesas".EstadoVI[#Mesa].Err_TOut_Avance_E1_E3 := TRUE;
   END_IF;
   IF "DB900_Estado_Mesas".EstadoVI[#Mesa].Err_TOut_Avance_E1_E3 THEN
       "DB900_Estado_Mesas".EstadoVI[#Mesa].Error_Mx := TRUE;
   END_IF;
END_REGION

REGION Network 20
   RUNG wire#powerrail
      "FC911_CNT_Tiempo_UHS"(Temporizar := wire#w1, Valor_Tiempo := #V_TOut_TR, Base_tiempo_ms := 1, Valor_Actual := "DB230_CONTADORES".Mesa[#Mesa].CNT_Bloqueo_Movimiento, Tiempo_OK => #tout_transfer)
   END_RUNG
   RUNG wire#powerrail
      Contact( #TEMP_MA_TR_Pos_E1 )
      I_Contact( #PosTR_E1 )
   END_RUNG wire#w1
   RUNG wire#powerrail
      Contact( #TEMP_MA_TR_Pos_S2 )
      I_Contact( #PosTR_S2 )
   END_RUNG wire#w1
   // the same network as SCL:
   "FC911_CNT_Tiempo_UHS"(Temporizar := (#TEMP_MA_TR_Pos_E1 AND NOT #PosTR_E1) OR (#TEMP_MA_TR_Pos_S2 AND NOT #PosTR_S2),
                          Valor_Tiempo := #V_TOut_TR,
                          Base_tiempo_ms := 1,
                          Valor_Actual := "DB230_CONTADORES".Mesa[#Mesa].CNT_Bloqueo_Movimiento,
                          Tiempo_OK => #tout_transfer);
END_REGION

REGION Network 21: Marca General Error
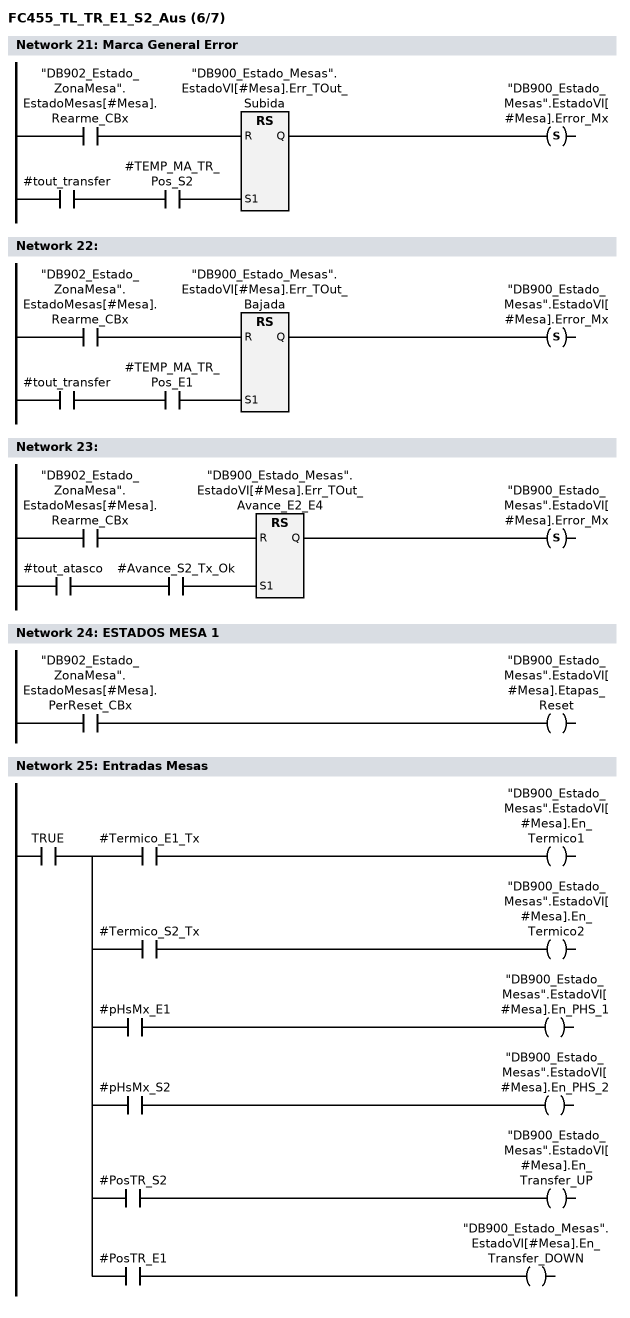
   RUNG wire#powerrail
      Contact( "DB902_Estado_ZonaMesa".EstadoMesas[#Mesa].Rearme_CBx )
      S_RS(operand := "DB900_Estado_Mesas".EstadoVI[#Mesa].Err_TOut_Subida, s1 := wire#w1)
      S_Coil( "DB900_Estado_Mesas".EstadoVI[#Mesa].Error_Mx )
   END_RUNG
   RUNG wire#powerrail
      Contact( #tout_transfer )
      Contact( #TEMP_MA_TR_Pos_S2 )
   END_RUNG wire#w1
   // the same network as SCL:
   IF "DB902_Estado_ZonaMesa".EstadoMesas[#Mesa].Rearme_CBx THEN
       "DB900_Estado_Mesas".EstadoVI[#Mesa].Err_TOut_Subida := FALSE;   // RS flip-flop
   END_IF;
   IF #tout_transfer AND #TEMP_MA_TR_Pos_S2 THEN
       "DB900_Estado_Mesas".EstadoVI[#Mesa].Err_TOut_Subida := TRUE;
   END_IF;
   IF "DB900_Estado_Mesas".EstadoVI[#Mesa].Err_TOut_Subida THEN
       "DB900_Estado_Mesas".EstadoVI[#Mesa].Error_Mx := TRUE;
   END_IF;
END_REGION

REGION Network 22
   RUNG wire#powerrail
      Contact( "DB902_Estado_ZonaMesa".EstadoMesas[#Mesa].Rearme_CBx )
      S_RS(operand := "DB900_Estado_Mesas".EstadoVI[#Mesa].Err_TOut_Bajada, s1 := wire#w1)
      S_Coil( "DB900_Estado_Mesas".EstadoVI[#Mesa].Error_Mx )
   END_RUNG
   RUNG wire#powerrail
      Contact( #tout_transfer )
      Contact( #TEMP_MA_TR_Pos_E1 )
   END_RUNG wire#w1
   // the same network as SCL:
   IF "DB902_Estado_ZonaMesa".EstadoMesas[#Mesa].Rearme_CBx THEN
       "DB900_Estado_Mesas".EstadoVI[#Mesa].Err_TOut_Bajada := FALSE;   // RS flip-flop
   END_IF;
   IF #tout_transfer AND #TEMP_MA_TR_Pos_E1 THEN
       "DB900_Estado_Mesas".EstadoVI[#Mesa].Err_TOut_Bajada := TRUE;
   END_IF;
   IF "DB900_Estado_Mesas".EstadoVI[#Mesa].Err_TOut_Bajada THEN
       "DB900_Estado_Mesas".EstadoVI[#Mesa].Error_Mx := TRUE;
   END_IF;
END_REGION

REGION Network 23
   RUNG wire#powerrail
      Contact( "DB902_Estado_ZonaMesa".EstadoMesas[#Mesa].Rearme_CBx )
      S_RS(operand := "DB900_Estado_Mesas".EstadoVI[#Mesa].Err_TOut_Avance_E2_E4, s1 := wire#w1)
      S_Coil( "DB900_Estado_Mesas".EstadoVI[#Mesa].Error_Mx )
   END_RUNG
   RUNG wire#powerrail
      Contact( #tout_atasco )
      Contact( #Avance_S2_Tx_Ok )
   END_RUNG wire#w1
   // the same network as SCL:
   IF "DB902_Estado_ZonaMesa".EstadoMesas[#Mesa].Rearme_CBx THEN
       "DB900_Estado_Mesas".EstadoVI[#Mesa].Err_TOut_Avance_E2_E4 := FALSE;   // RS flip-flop
   END_IF;
   IF #tout_atasco AND #Avance_S2_Tx_Ok THEN
       "DB900_Estado_Mesas".EstadoVI[#Mesa].Err_TOut_Avance_E2_E4 := TRUE;
   END_IF;
   IF "DB900_Estado_Mesas".EstadoVI[#Mesa].Err_TOut_Avance_E2_E4 THEN
       "DB900_Estado_Mesas".EstadoVI[#Mesa].Error_Mx := TRUE;
   END_IF;
END_REGION

REGION Network 24: ESTADOS MESA 1
   RUNG wire#powerrail
      Contact( "DB902_Estado_ZonaMesa".EstadoMesas[#Mesa].PerReset_CBx )
      Coil( "DB900_Estado_Mesas".EstadoVI[#Mesa].Etapas_Reset )
   END_RUNG
   // the same network as SCL:
   "DB900_Estado_Mesas".EstadoVI[#Mesa].Etapas_Reset := "DB902_Estado_ZonaMesa".EstadoMesas[#Mesa].PerReset_CBx;
END_REGION

REGION Network 25: Entradas Mesas
   RUNG wire#powerrail
      Contact( TRUE )
      wire#w1
      Contact( #Termico_E1_Tx )
      Coil( "DB900_Estado_Mesas".EstadoVI[#Mesa].En_Termico1 )
   END_RUNG
   RUNG wire#w1
      Contact( #Termico_S2_Tx )
      Coil( "DB900_Estado_Mesas".EstadoVI[#Mesa].En_Termico2 )
   END_RUNG
   RUNG wire#w1
      Contact( #pHsMx_E1 )
      Coil( "DB900_Estado_Mesas".EstadoVI[#Mesa].En_PHS_1 )
   END_RUNG
   RUNG wire#w1
      Contact( #pHsMx_S2 )
      Coil( "DB900_Estado_Mesas".EstadoVI[#Mesa].En_PHS_2 )
   END_RUNG
   RUNG wire#w1
      Contact( #PosTR_S2 )
      Coil( "DB900_Estado_Mesas".EstadoVI[#Mesa].En_Transfer_UP )
   END_RUNG
   RUNG wire#w1
      Contact( #PosTR_E1 )
      Coil( "DB900_Estado_Mesas".EstadoVI[#Mesa].En_Transfer_DOWN )
   END_RUNG
   // the same network as SCL:
   "DB900_Estado_Mesas".EstadoVI[#Mesa].En_Termico1 := TRUE AND #Termico_E1_Tx;
   "DB900_Estado_Mesas".EstadoVI[#Mesa].En_Termico2 := TRUE AND #Termico_S2_Tx;
   "DB900_Estado_Mesas".EstadoVI[#Mesa].En_PHS_1 := TRUE AND #pHsMx_E1;
   "DB900_Estado_Mesas".EstadoVI[#Mesa].En_PHS_2 := TRUE AND #pHsMx_S2;
   "DB900_Estado_Mesas".EstadoVI[#Mesa].En_Transfer_UP := TRUE AND #PosTR_S2;
   "DB900_Estado_Mesas".EstadoVI[#Mesa].En_Transfer_DOWN := TRUE AND #PosTR_E1;
END_REGION

REGION Network 26: Salidas Mesas
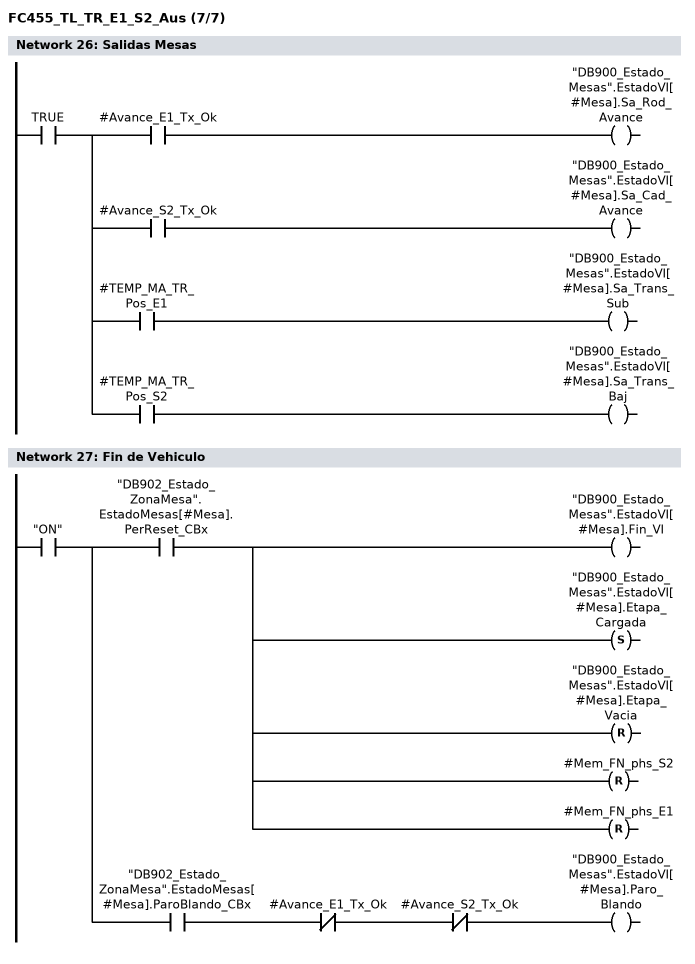
   RUNG wire#powerrail
      Contact( TRUE )
      wire#w1
      Contact( #Avance_E1_Tx_Ok )
      Coil( "DB900_Estado_Mesas".EstadoVI[#Mesa].Sa_Rod_Avance )
   END_RUNG
   RUNG wire#w1
      Contact( #Avance_S2_Tx_Ok )
      Coil( "DB900_Estado_Mesas".EstadoVI[#Mesa].Sa_Cad_Avance )
   END_RUNG
   RUNG wire#w1
      Contact( #TEMP_MA_TR_Pos_E1 )
      Coil( "DB900_Estado_Mesas".EstadoVI[#Mesa].Sa_Trans_Sub )
   END_RUNG
   RUNG wire#w1
      Contact( #TEMP_MA_TR_Pos_S2 )
      Coil( "DB900_Estado_Mesas".EstadoVI[#Mesa].Sa_Trans_Baj )
   END_RUNG
   // the same network as SCL:
   "DB900_Estado_Mesas".EstadoVI[#Mesa].Sa_Rod_Avance := TRUE AND #Avance_E1_Tx_Ok;
   "DB900_Estado_Mesas".EstadoVI[#Mesa].Sa_Cad_Avance := TRUE AND #Avance_S2_Tx_Ok;
   "DB900_Estado_Mesas".EstadoVI[#Mesa].Sa_Trans_Sub := TRUE AND #TEMP_MA_TR_Pos_E1;
   "DB900_Estado_Mesas".EstadoVI[#Mesa].Sa_Trans_Baj := TRUE AND #TEMP_MA_TR_Pos_S2;
END_REGION

REGION Network 27: Fin de Vehiculo
   RUNG wire#powerrail
      Contact( "ON" )
      wire#w1
      Contact( "DB902_Estado_ZonaMesa".EstadoMesas[#Mesa].PerReset_CBx )
      wire#w2
      Coil( "DB900_Estado_Mesas".EstadoVI[#Mesa].Fin_VI )
   END_RUNG
   RUNG wire#w2
      S_Coil( "DB900_Estado_Mesas".EstadoVI[#Mesa].Etapa_Cargada )
   END_RUNG
   RUNG wire#w2
      R_Coil( "DB900_Estado_Mesas".EstadoVI[#Mesa].Etapa_Vacia )
   END_RUNG
   RUNG wire#w2
      R_Coil( #Mem_FN_phs_S2 )
   END_RUNG
   RUNG wire#w2
      R_Coil( #Mem_FN_phs_E1 )
   END_RUNG
   RUNG wire#w1
      Contact( "DB902_Estado_ZonaMesa".EstadoMesas[#Mesa].ParoBlando_CBx )
      I_Contact( #Avance_E1_Tx_Ok )
      I_Contact( #Avance_S2_Tx_Ok )
      Coil( "DB900_Estado_Mesas".EstadoVI[#Mesa].Paro_Blando )
   END_RUNG
   // the same network as SCL:
   #_w1 := "ON" AND "DB902_Estado_ZonaMesa".EstadoMesas[#Mesa].PerReset_CBx;
   "DB900_Estado_Mesas".EstadoVI[#Mesa].Fin_VI := "ON" AND "DB902_Estado_ZonaMesa".EstadoMesas[#Mesa].PerReset_CBx;
   IF #_w1 THEN
       "DB900_Estado_Mesas".EstadoVI[#Mesa].Etapa_Cargada := TRUE;
       "DB900_Estado_Mesas".EstadoVI[#Mesa].Etapa_Vacia := FALSE;
       #Mem_FN_phs_S2 := FALSE;
       #Mem_FN_phs_E1 := FALSE;
   END_IF;
   "DB900_Estado_Mesas".EstadoVI[#Mesa].Paro_Blando := "ON" AND "DB902_Estado_ZonaMesa".EstadoMesas[#Mesa].ParoBlando_CBx AND NOT #Avance_E1_Tx_Ok AND NOT #Avance_S2_Tx_Ok;
END_REGION
END_FUNCTION
